(* Logix 5000 project; controller NSH_PLC1 vendor 1 type 14 code 167 rev 32.11; software revision 32.02; part 11 of 12 *)
(* tags used below, declared in another part *)
   Num_Faults : DINT;   // Number of PreCelan Faults
   Num_Warnings : DINT;   // Number of PreCelan Warnings
   Reset_TOF_PRE : DINT;   // Reset pulse duration to Drives
   SpeedIsFactored : BOOL;   // Speed of VFD is factored by Master Speed Factor
   TempAccelerating : BOOL;   // Temp Motor is Accelerating
   TempActive : BOOL;   // Temp Motor is Active
   TempAlarm : BOOL;   // Temp Motor has Alarm
   TempAtSpeed : BOOL;   // Temp Motor is At Speed
   TempCommAlarm : BOOL;   // Temp Motor, AOP communications Alarm
   TempDecelerating : BOOL;   // Temp Motor is Decelerating
   TempFaulted : BOOL;   // Temp Motor is Faulted
   TempMotor : Motor;
   TempReady : BOOL;   // Temp Motor is ready
   TempRunning : BOOL;   // Temp Motor is Running
   TempVFD : VFD_Extra;   // Temp VFD Structure
   BH_FansStarting : BOOL;   // Baghouse 1, 2 or 3 Fans Starting
   CR_LastLine1 : BOOL;   // Last Motor in line 1 Running
   CR_LastLine2 : BOOL;   // Last Motor in line 2 Running
   CR_LastPC1Fan : BOOL;   // Last Motor in Line 1 Fans Running
   CR_LastPC2Fan : BOOL;   // Last Motor in Line 2 Fans Running
   CR_RunCommon : BOOL;   // PreClean, Run Common Units
   CR_RunLine1 : BOOL;   // Pre Clean Run Line 1 Relay
   CR_RunLine2 : BOOL;   // Pre Clean Run Line 2 Relay
   CR_RunPC1_Fans : BOOL;   // Pre Clean Run Line 1 Fans Relay
   CR_RunPC1_FansCO : BOOL;   // Pre Clean Run Line 1 Fans Cleanout Relay
   CR_RunPC2_Fans : BOOL;   // Pre Clean Run Line 2 Fans Relay
   CR_RunPC2_FansCO : BOOL;   // Pre Clean Run Line 2 Fans Cleanout Relay
   CR_StopCommon : BOOL;   // PreClean, Stop Common Units
   CR_StopLine1 : BOOL;   // Pre Clean Stop Line 1 Relay
   CR_StopLine2 : BOOL;   // Pre Clean Stop Line 2 Relay
   DummyVFD : VFD_Extra;   // Dummy
   HS_Starting : BOOL;   // Sheller Sequence is Starting, Prevent Preclean from Starting
   P10_5A : Motor;   // Cross Auger
   P10_5B : Motor;   // Cross Auger
   P10A : Motor;   // Elev to Bins
   P10B : Motor;   // Elev to Bins
   P11A : Motor;   // Line1 Auger
   P11B : Motor;   // Line2 Auger
   P1A : Motor;   // DO Conv.
   P1B : Motor;   // Auger
   P2A : Motor;   // Cross Conv.
   P2B : Motor;   // Stick Reel
   P3A : Motor;   // Stick Reel
   P3B : Motor;   // Stick Reel
   P4A : Motor;   // C. Belt
   P4B : Motor;   // C. Belt
   P5A : Motor;   // Ele. to Vib
   P5B : Motor;   // Ele. to Vib
   P6A : Motor;   // Vib Splitter
   P6B : Motor;   // Vib.Spltr.
   P7A1 : Motor;   // Screener
   P7A2 : Motor;   // Screener
   P7B : Motor;   // Screener
   P7B2_A : Motor;   // Screener
   P7B2_B : Motor;   // Rot.Fdr.
   P8A2_A : Motor;   // Destoner
   P8A2_B : Motor;   // AirLock
   P8A_A : Motor;   // Destoner
   P8A_B : Motor;   // Airlock
   P8B : Motor;   // Destoner
   P8B2_A : Motor;   // Destoner
   P8B2_B : Motor;   // Rot.Fdr.
   P9A : Motor;   // Auger
   P9B : Motor;   // Auger
   PB_StartLine1 : BOOL;   // Pre Clean Start Line 1 Button
   PB_StartLine2 : BOOL;   // Pre Clean Start Line 2 Button
   PB_StopLine1 : BOOL;   // Pre Clean Stop Line 1 Button
   PB_StopLine2 : BOOL;   // Pre Clean Stop Line 2 Button
   PBB1A : Motor;   // AirLock
   PBB1B : Motor;   // Arm
   PBB1C : Motor;   // Cleaning Fan,
   PBB1D : Motor;   // Fan,
   PBB1D_VFD : VFD_Extra;   // Fan
   PBB2A : Motor;   // AirLock
   PBB2B : Motor;   // Arm
   PBB2C : Motor;   // Cleaning Fan,
   PBB2D : Motor;   // Fan,
   PBL_StartLine1 : BOOL;   // Pre Clean Start Line 1 Button Light
   PBL_StartLine2 : BOOL;   // Pre Clean Start Line 2 Button Light
   PBL_StopLine1 : BOOL;   // Pre Clean Stop Line 1 Button Light
   PBL_StopLine2 : BOOL;   // Pre Clean Stop Line 2 Button Light
   PC_AlarmPulseHorn : BOOL;   // PreClean, New Alarm, Pulse Horn
   PC_FaultResetHorn : BOOL;   // PreClean, Fault Reset, sound Horn
   PC_Horn : BOOL;   // PreClean, Horn Output
   PC_LinesStarting : BOOL;   // Pre Clean Line 1 or 2 Starting
   PC_NoEstops : BOOL;   // PreClean, No Estops
   PD1 : Motor;   // Dirt Conv.
   PD2 : Motor;   // Incline
   PR1 : Motor;   // Rock Conv.
   PR2 : Motor;   // Inc. Rock
   PR3 : Motor;   // Belt
   PS1 : Motor;   // Stick Conv.
   PS2 : Motor;   // Inc. Stick Conv.
   PS3 : Motor;   // Twig Conv.
   PS4 : Motor;   // Twig Conv.
   TMR_LineStart1 : TIMER;   // Pre Clean Line 1 Start Warning Timer
   TMR_LineStart2 : TIMER;   // Pre Clean Line 2 Start Warning Timer
   TMR_StartPC1_Fans : TIMER;   // Pre Clean Line 1 Fans Start Warning Timer
   TMR_StartPC1_FansCO : TIMER;   // Pre Clean Line 1 Fans Cleanout Start Warning Timer
   TMR_StartPC2_Fans : TIMER;   // Pre Clean Line 2 Fans Start Warning Timer
   TMR_StartPC2_FansCO : TIMER;   // Pre Clean Line 2 Fans Cleanout Start Warning Timer
(* PreClean, continued *)

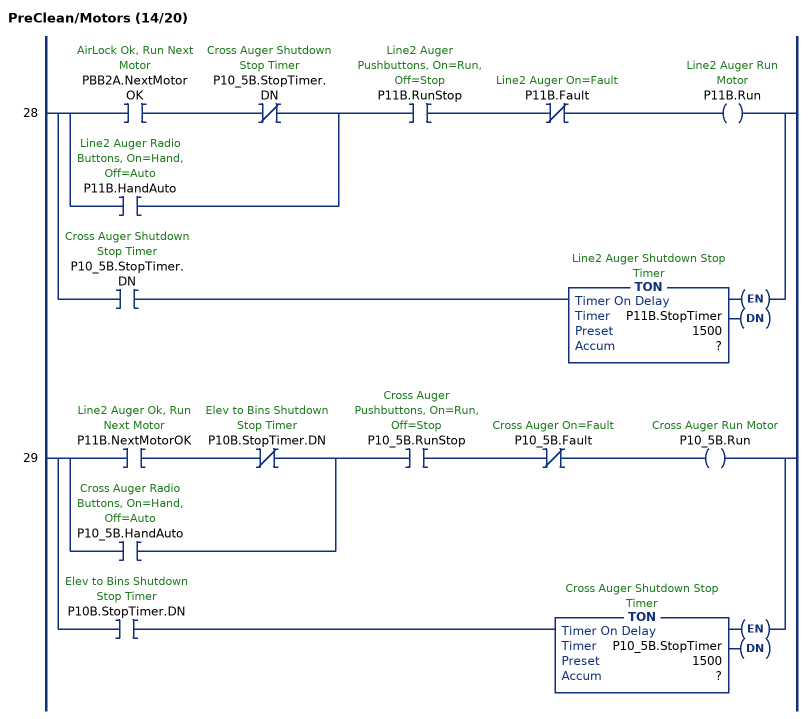
   28: [[XIC(PBB2A.NextMotorOK) XIO(P10_5B.StopTimer.DN) ,XIC(P11B.HandAuto) ] XIC(P11B.RunStop) XIO(P11B.Fault) OTE(P11B.Run) ,XIC(P10_5B.StopTimer.DN) TON(P11B.StopTimer,?,?) ];
   29: [[XIC(P11B.NextMotorOK) XIO(P10B.StopTimer.DN) ,XIC(P10_5B.HandAuto) ] XIC(P10_5B.RunStop) XIO(P10_5B.Fault) OTE(P10_5B.Run) ,XIC(P10B.StopTimer.DN) TON(P10_5B.StopTimer,?,?) ];
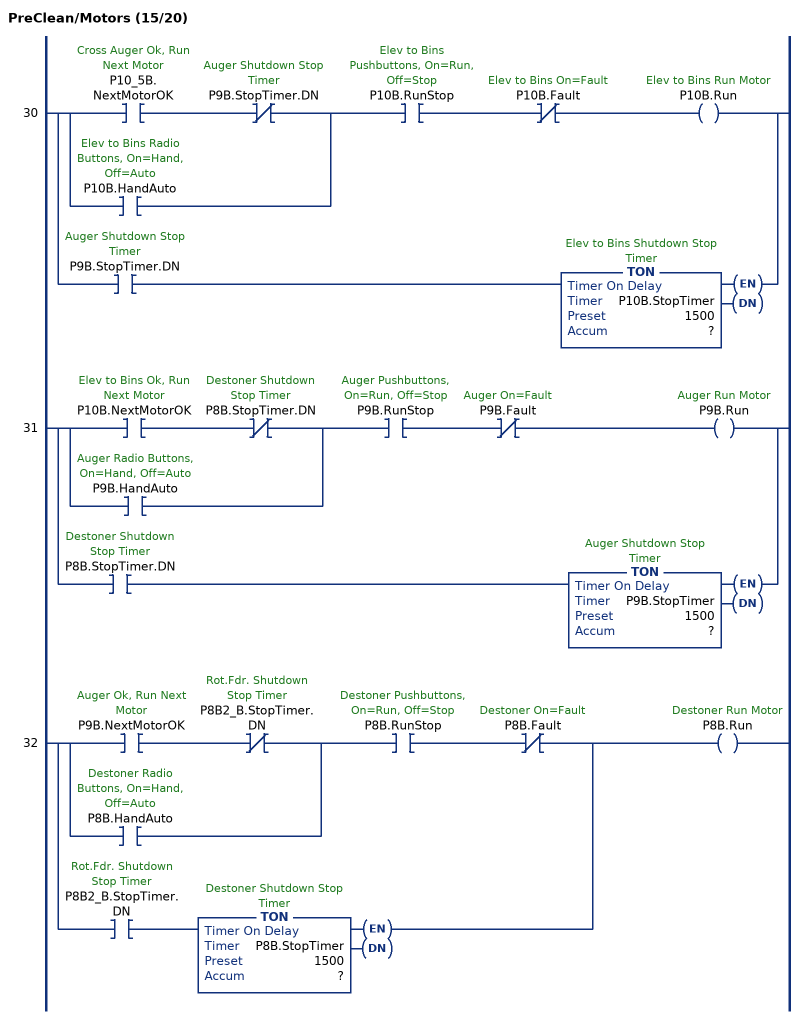
   30: [[XIC(P10_5B.NextMotorOK) XIO(P9B.StopTimer.DN) ,XIC(P10B.HandAuto) ] XIC(P10B.RunStop) XIO(P10B.Fault) OTE(P10B.Run) ,XIC(P9B.StopTimer.DN) TON(P10B.StopTimer,?,?) ];
   31: [[XIC(P10B.NextMotorOK) XIO(P8B.StopTimer.DN) ,XIC(P9B.HandAuto) ] XIC(P9B.RunStop) XIO(P9B.Fault) OTE(P9B.Run) ,XIC(P8B.StopTimer.DN) TON(P9B.StopTimer,?,?) ];
   32: [[XIC(P9B.NextMotorOK) XIO(P8B2_B.StopTimer.DN) ,XIC(P8B.HandAuto) ] XIC(P8B.RunStop) XIO(P8B.Fault) ,XIC(P8B2_B.StopTimer.DN) TON(P8B.StopTimer,?,?) ]OTE(P8B.Run);
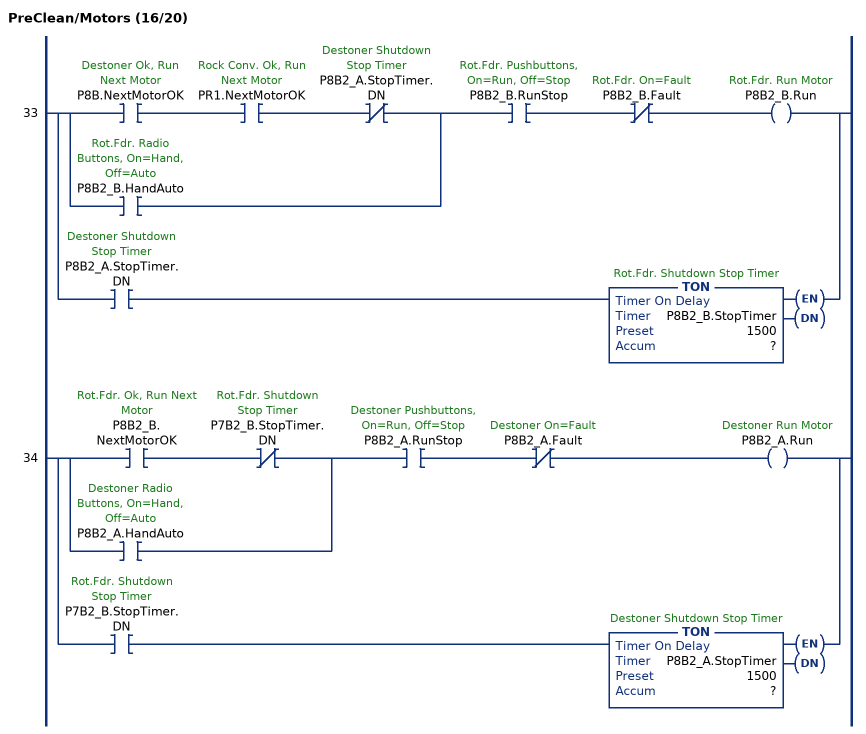
   33: [[XIC(P8B.NextMotorOK) XIC(PR1.NextMotorOK) XIO(P8B2_A.StopTimer.DN) ,XIC(P8B2_B.HandAuto) ] XIC(P8B2_B.RunStop) XIO(P8B2_B.Fault) OTE(P8B2_B.Run) ,XIC(P8B2_A.StopTimer.DN) TON(P8B2_B.StopTimer,?,?) ];
   34: [[XIC(P8B2_B.NextMotorOK) XIO(P7B2_B.StopTimer.DN) ,XIC(P8B2_A.HandAuto) ] XIC(P8B2_A.RunStop) XIO(P8B2_A.Fault) OTE(P8B2_A.Run) ,XIC(P7B2_B.StopTimer.DN) TON(P8B2_A.StopTimer,?,?) ];
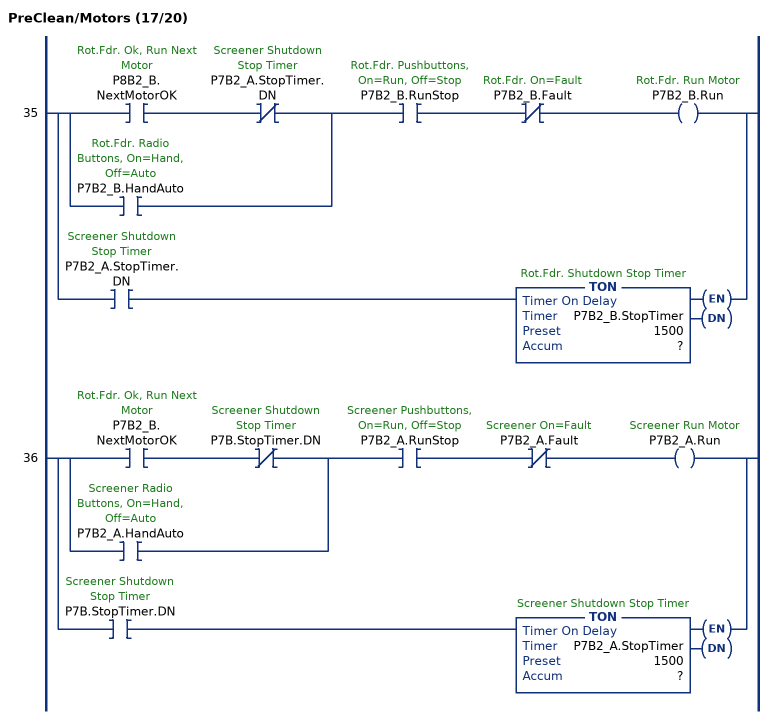
   35: [[XIC(P8B2_B.NextMotorOK) XIO(P7B2_A.StopTimer.DN) ,XIC(P7B2_B.HandAuto) ] XIC(P7B2_B.RunStop) XIO(P7B2_B.Fault) OTE(P7B2_B.Run) ,XIC(P7B2_A.StopTimer.DN) TON(P7B2_B.StopTimer,?,?) ];
   36: [[XIC(P7B2_B.NextMotorOK) XIO(P7B.StopTimer.DN) ,XIC(P7B2_A.HandAuto) ] XIC(P7B2_A.RunStop) XIO(P7B2_A.Fault) OTE(P7B2_A.Run) ,XIC(P7B.StopTimer.DN) TON(P7B2_A.StopTimer,?,?) ];
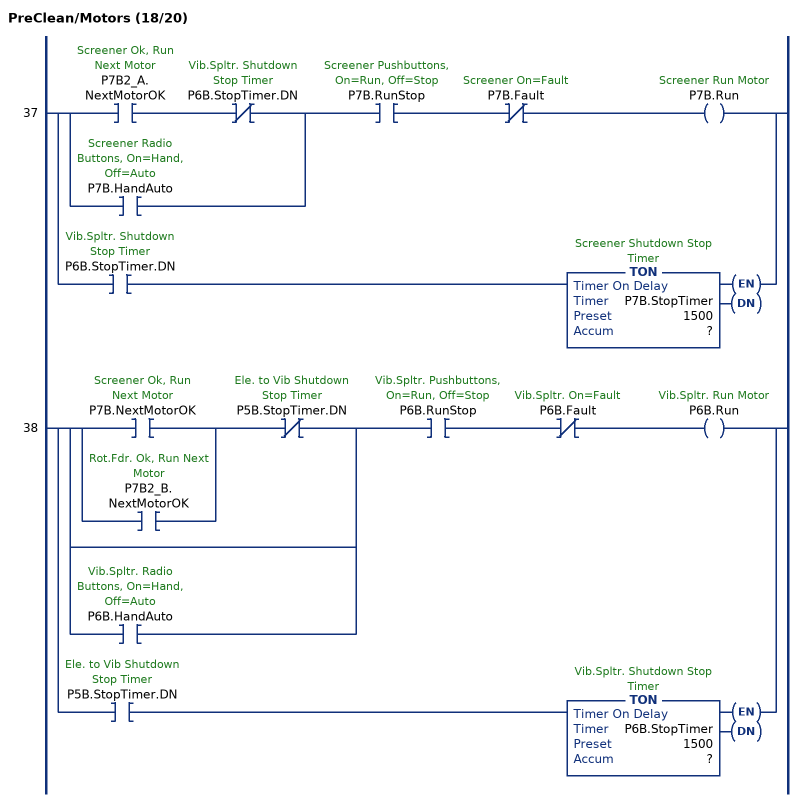
   37: [[XIC(P7B2_A.NextMotorOK) XIO(P6B.StopTimer.DN) ,XIC(P7B.HandAuto) ] XIC(P7B.RunStop) XIO(P7B.Fault) OTE(P7B.Run) ,XIC(P6B.StopTimer.DN) TON(P7B.StopTimer,?,?) ];
   38: [[[XIC(P7B.NextMotorOK) ,XIC(P7B2_B.NextMotorOK) ] XIO(P5B.StopTimer.DN) ,,XIC(P6B.HandAuto) ] XIC(P6B.RunStop) XIO(P6B.Fault) OTE(P6B.Run) ,XIC(P5B.StopTimer.DN) TON(P6B.StopTimer,?,?) ];
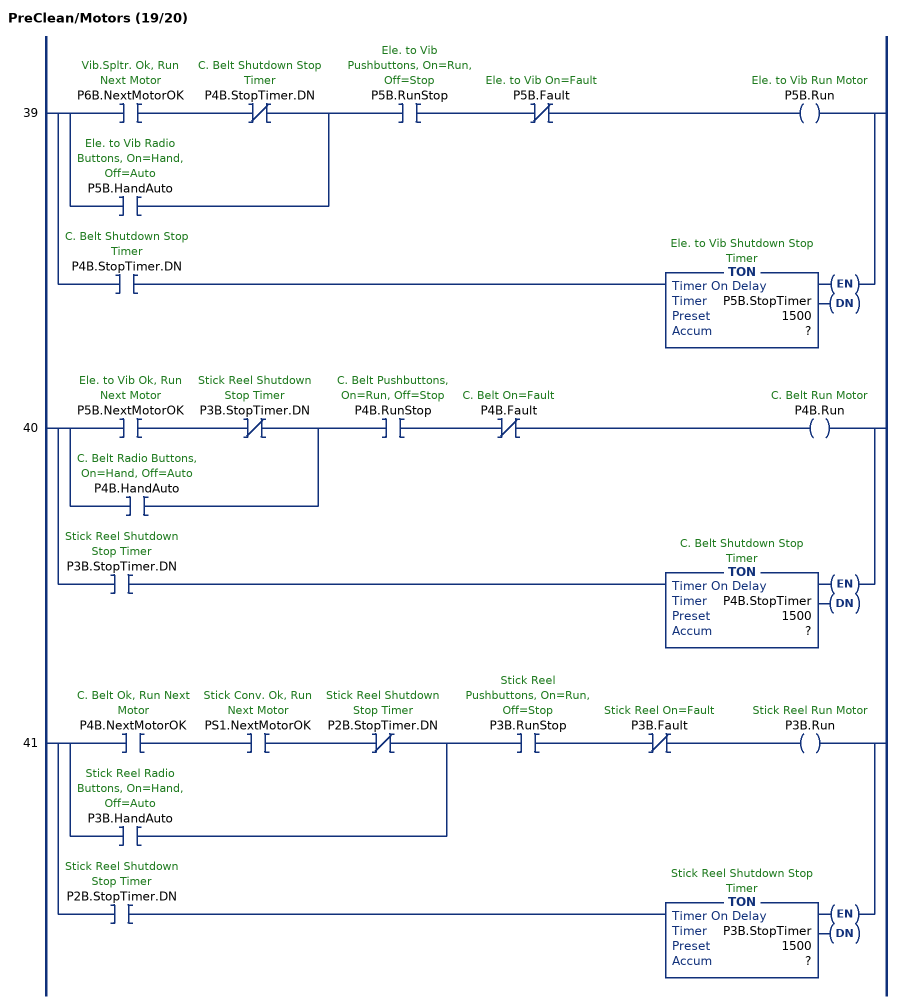
   39: [[XIC(P6B.NextMotorOK) XIO(P4B.StopTimer.DN) ,XIC(P5B.HandAuto) ] XIC(P5B.RunStop) XIO(P5B.Fault) OTE(P5B.Run) ,XIC(P4B.StopTimer.DN) TON(P5B.StopTimer,?,?) ];
   40: [[XIC(P5B.NextMotorOK) XIO(P3B.StopTimer.DN) ,XIC(P4B.HandAuto) ] XIC(P4B.RunStop) XIO(P4B.Fault) OTE(P4B.Run) ,XIC(P3B.StopTimer.DN) TON(P4B.StopTimer,?,?) ];
   41: [[XIC(P4B.NextMotorOK) XIC(PS1.NextMotorOK) XIO(P2B.StopTimer.DN) ,XIC(P3B.HandAuto) ] XIC(P3B.RunStop) XIO(P3B.Fault) OTE(P3B.Run) ,XIC(P2B.StopTimer.DN) TON(P3B.StopTimer,?,?) ];
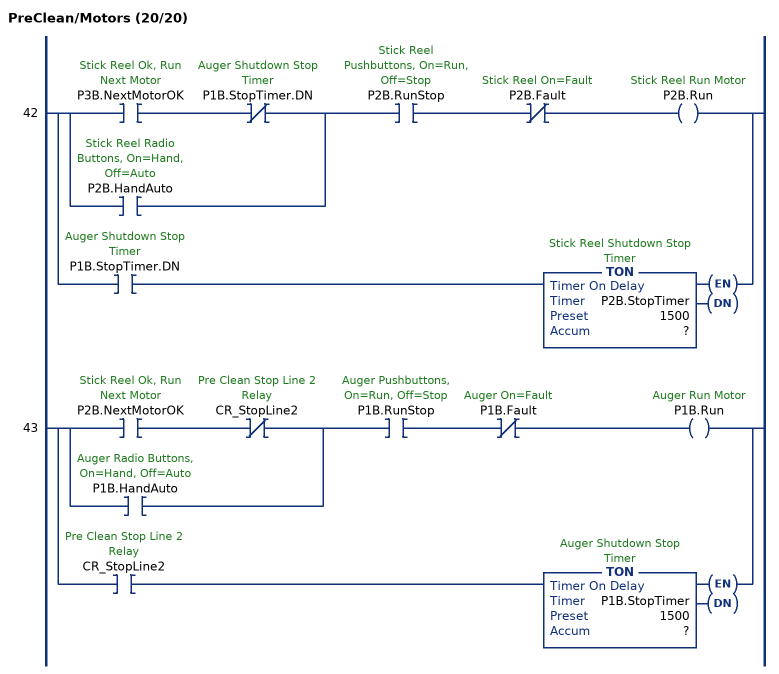
   42: [[XIC(P3B.NextMotorOK) XIO(P1B.StopTimer.DN) ,XIC(P2B.HandAuto) ] XIC(P2B.RunStop) XIO(P2B.Fault) OTE(P2B.Run) ,XIC(P1B.StopTimer.DN) TON(P2B.StopTimer,?,?) ];
   43: [[XIC(P2B.NextMotorOK) XIO(CR_StopLine2) ,XIC(P1B.HandAuto) ] XIC(P1B.RunStop) XIO(P1B.Fault) OTE(P1B.Run) ,XIC(CR_StopLine2) TON(P1B.StopTimer,?,?) ];
END_ROUTINE

ROUTINE MotorStatusSUB   (* ladder *)
// Update Status Subroutine
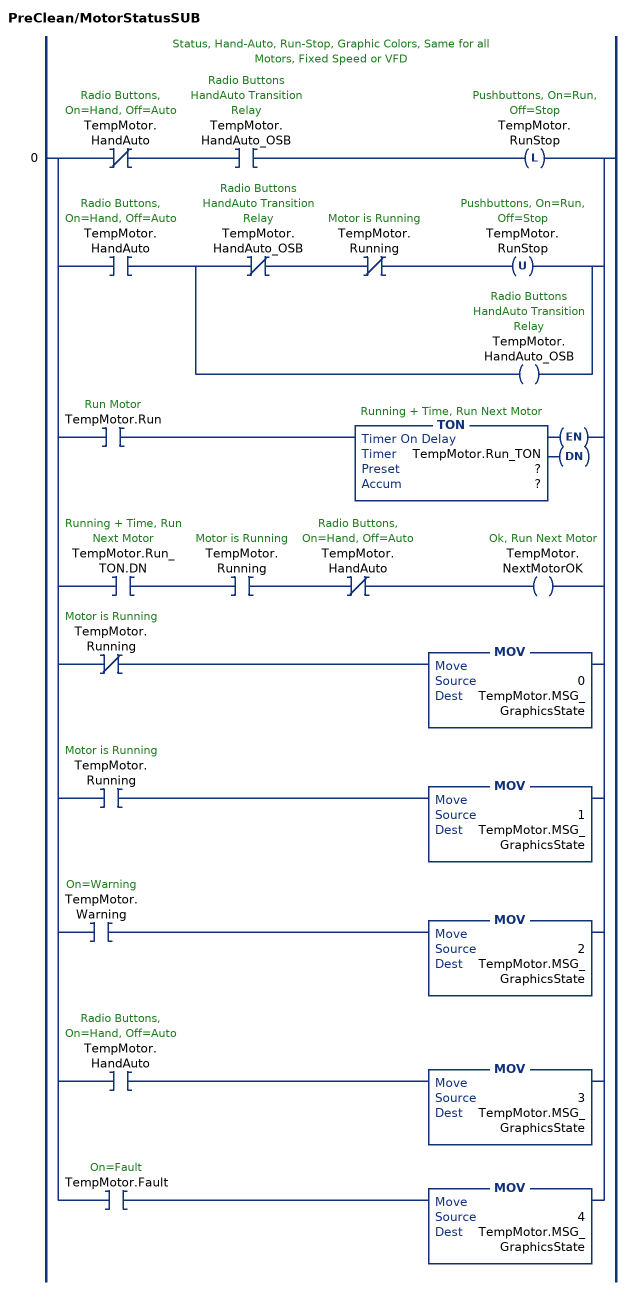
   // Status, Hand-Auto, Run-Stop, Graphic Colors, Same for all
   // Motors, Fixed Speed or VFD
   0: [XIO(TempMotor.HandAuto) XIC(TempMotor.HandAuto_OSB) OTL(TempMotor.RunStop) ,XIC(TempMotor.HandAuto) [XIO(TempMotor.HandAuto_OSB) XIO(TempMotor.Running) OTU(TempMotor.RunStop) ,OTE(TempMotor.HandAuto_OSB) ] ,XIC(TempMotor.Run) TON(TempMotor.Run_TON,?,?) ,XIC(TempMotor.Run_TON.DN) XIC(TempMotor.Running) XIO(TempMotor.HandAuto) OTE(TempMotor.NextMotorOK) ,XIO(TempMotor.Running) MOV(0,TempMotor.MSG_GraphicsState) ,XIC(TempMotor.Running) MOV(1,TempMotor.MSG_GraphicsState) ,XIC(TempMotor.Warning) MOV(2,TempMotor.MSG_GraphicsState) ,XIC(TempMotor.HandAuto) MOV(3,TempMotor.MSG_GraphicsState) ,XIC(TempMotor.Fault) MOV(4,TempMotor.MSG_GraphicsState) ];
END_ROUTINE

ROUTINE PC_MainJSR   (* ladder *)
// Jump To Other Routines
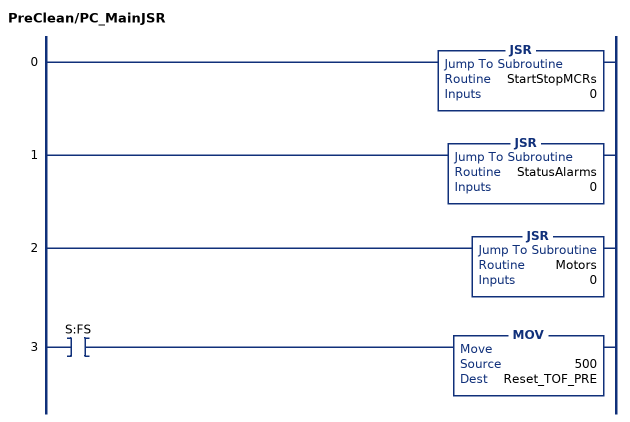
   0: JSR(StartStopMCRs,0);
   1: JSR(StatusAlarms,0);
   2: JSR(Motors,0);
   3: XIC(S:FS)MOV(500,Reset_TOF_PRE);
END_ROUTINE

ROUTINE PF525_StatusAlmWarnSUB   (* ladder *)
// Decode Status Bits and Set Warnings and Alarm for PowerFlex525
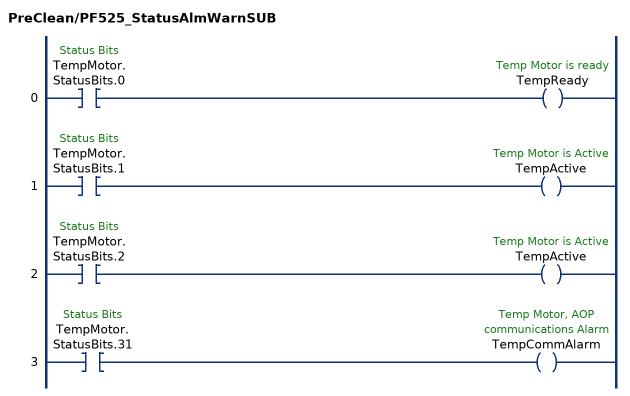
   0: XIC(TempMotor.StatusBits.0)OTE(TempReady);
   1: XIC(TempMotor.StatusBits.1)OTE(TempActive);
   2: XIC(TempMotor.StatusBits.2)OTE(TempActive);
   3: XIC(TempMotor.StatusBits.31)OTE(TempCommAlarm);
END_ROUTINE

ROUTINE PF755_StatusAlmWarnSUB   (* ladder *)
// Decode Status Bits and Set Warnings and Alarm for PowerFlex755
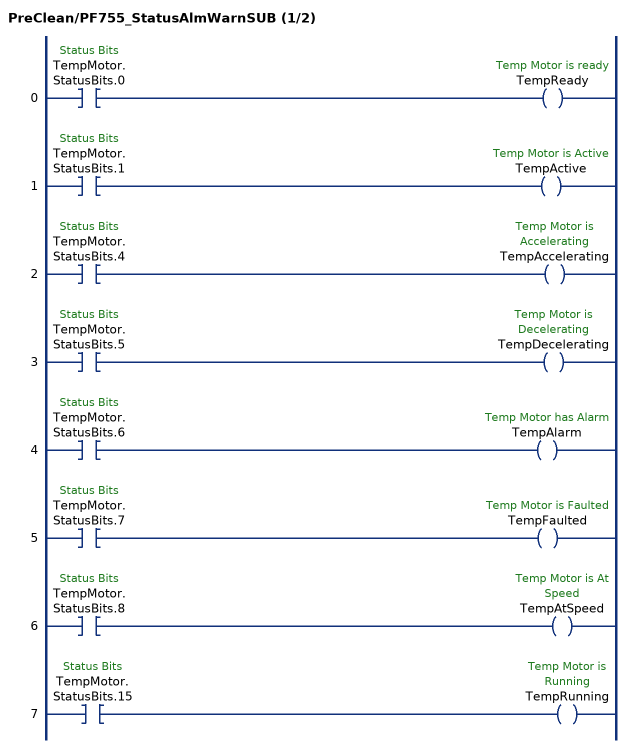
   0: XIC(TempMotor.StatusBits.0)OTE(TempReady);
   1: XIC(TempMotor.StatusBits.1)OTE(TempActive);
   2: XIC(TempMotor.StatusBits.4)OTE(TempAccelerating);
   3: XIC(TempMotor.StatusBits.5)OTE(TempDecelerating);
   4: XIC(TempMotor.StatusBits.6)OTE(TempAlarm);
   5: XIC(TempMotor.StatusBits.7)OTE(TempFaulted);
   6: XIC(TempMotor.StatusBits.8)OTE(TempAtSpeed);
   7: XIC(TempMotor.StatusBits.15)OTE(TempRunning);
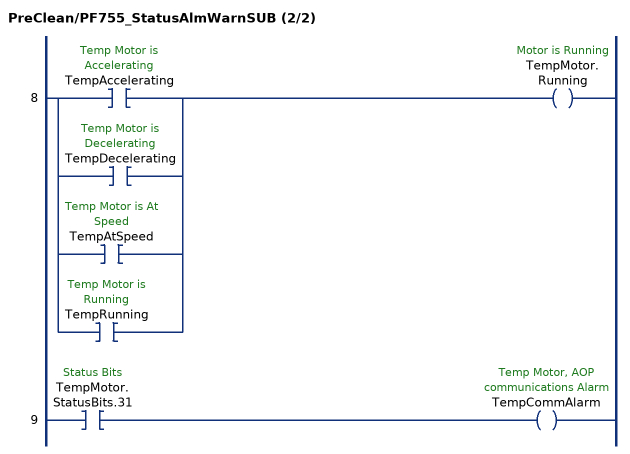
   8: [XIC(TempAccelerating) ,XIC(TempDecelerating) ,XIC(TempAtSpeed) ,XIC(TempRunning) ]OTE(TempMotor.Running);
   9: XIC(TempMotor.StatusBits.31)OTE(TempCommAlarm);
END_ROUTINE

ROUTINE StartStopMCRs   (* ladder *)
// Precleaner Logic
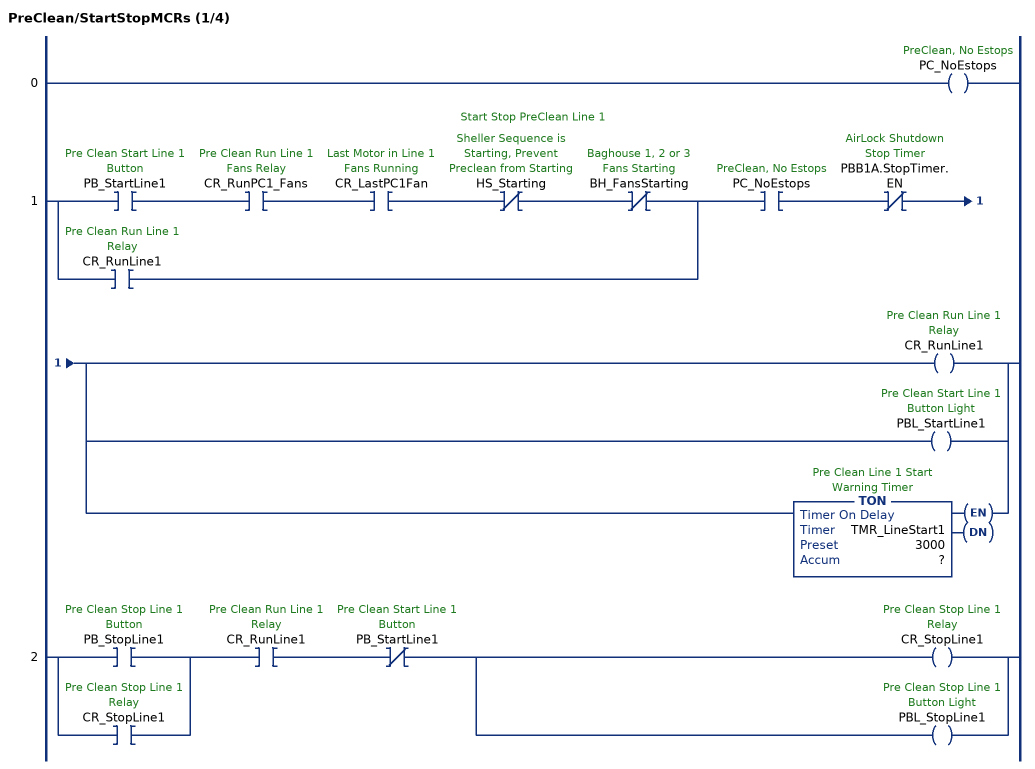
   0: OTE(PC_NoEstops);
   // Start Stop PreClean Line 1
   1: [XIC(PB_StartLine1) XIC(CR_RunPC1_Fans) XIC(CR_LastPC1Fan) XIO(HS_Starting) XIO(BH_FansStarting) ,XIC(CR_RunLine1) ]XIC(PC_NoEstops)XIO(PBB1A.StopTimer.EN)[OTE(CR_RunLine1) ,OTE(PBL_StartLine1) ,TON(TMR_LineStart1,?,?) ];
   2: [XIC(PB_StopLine1) ,XIC(CR_StopLine1) ]XIC(CR_RunLine1)XIO(PB_StartLine1)[OTE(CR_StopLine1) ,OTE(PBL_StopLine1) ];
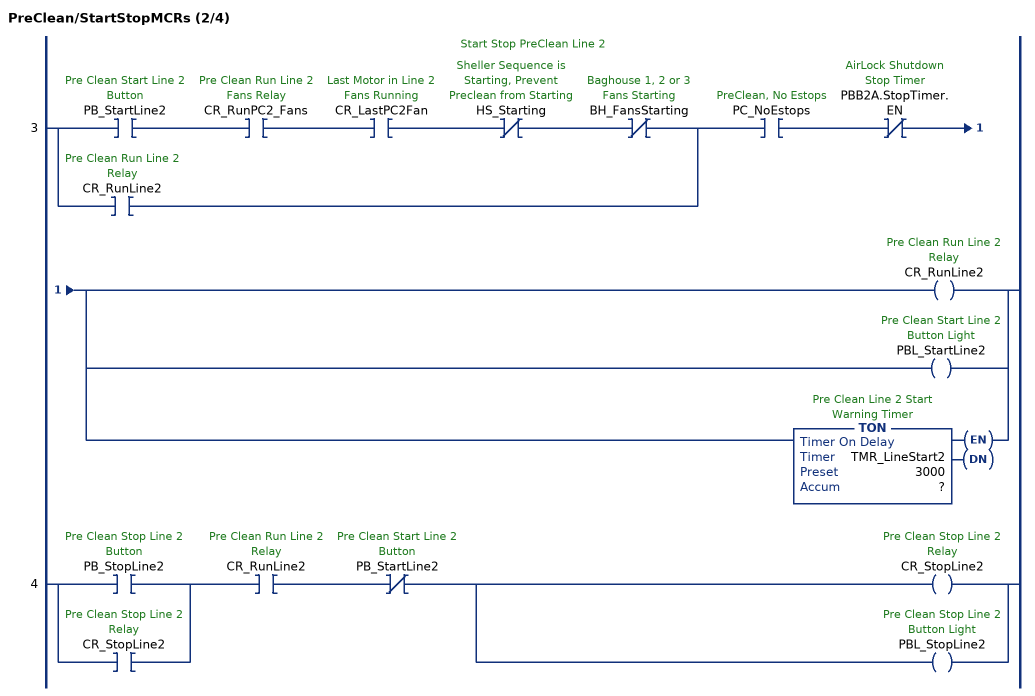
   // Start Stop PreClean Line 2
   3: [XIC(PB_StartLine2) XIC(CR_RunPC2_Fans) XIC(CR_LastPC2Fan) XIO(HS_Starting) XIO(BH_FansStarting) ,XIC(CR_RunLine2) ]XIC(PC_NoEstops)XIO(PBB2A.StopTimer.EN)[OTE(CR_RunLine2) ,OTE(PBL_StartLine2) ,TON(TMR_LineStart2,?,?) ];
   4: [XIC(PB_StopLine2) ,XIC(CR_StopLine2) ]XIC(CR_RunLine2)XIO(PB_StartLine2)[OTE(CR_StopLine2) ,OTE(PBL_StopLine2) ];
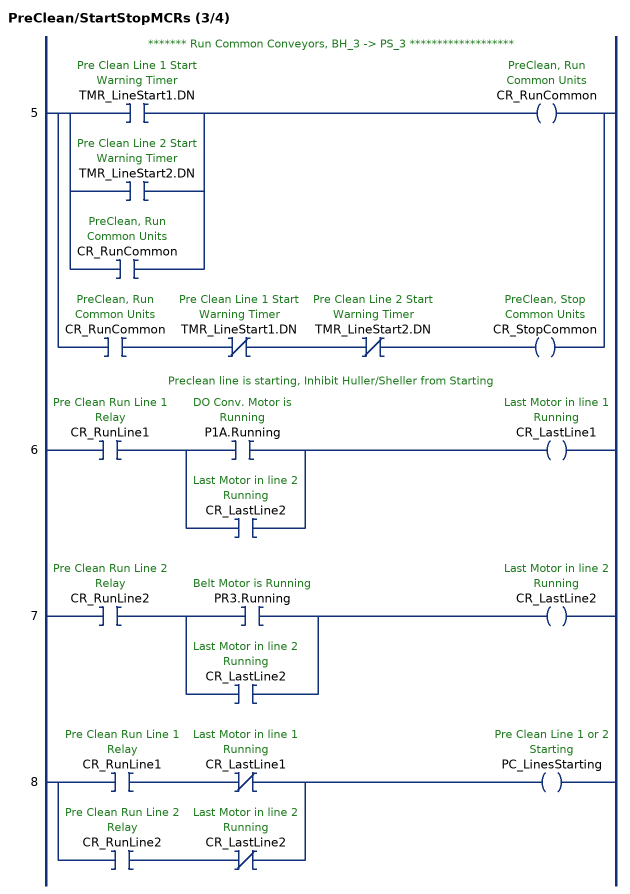
   // ******* Run Common Conveyors, BH_3 -> PS_3 *******************
   5: [[XIC(TMR_LineStart1.DN) ,XIC(TMR_LineStart2.DN) ,XIC(CR_RunCommon) ] OTE(CR_RunCommon) ,XIC(CR_RunCommon) XIO(TMR_LineStart1.DN) XIO(TMR_LineStart2.DN) OTE(CR_StopCommon) ];
   // Preclean line is starting, Inhibit Huller/Sheller from Starting
   6: XIC(CR_RunLine1)[XIC(P1A.Running) ,XIC(CR_LastLine2) ]OTE(CR_LastLine1);
   7: XIC(CR_RunLine2)[XIC(PR3.Running) ,XIC(CR_LastLine2) ]OTE(CR_LastLine2);
   8: [XIC(CR_RunLine1) XIO(CR_LastLine1) ,XIC(CR_RunLine2) XIO(CR_LastLine2) ]OTE(PC_LinesStarting);
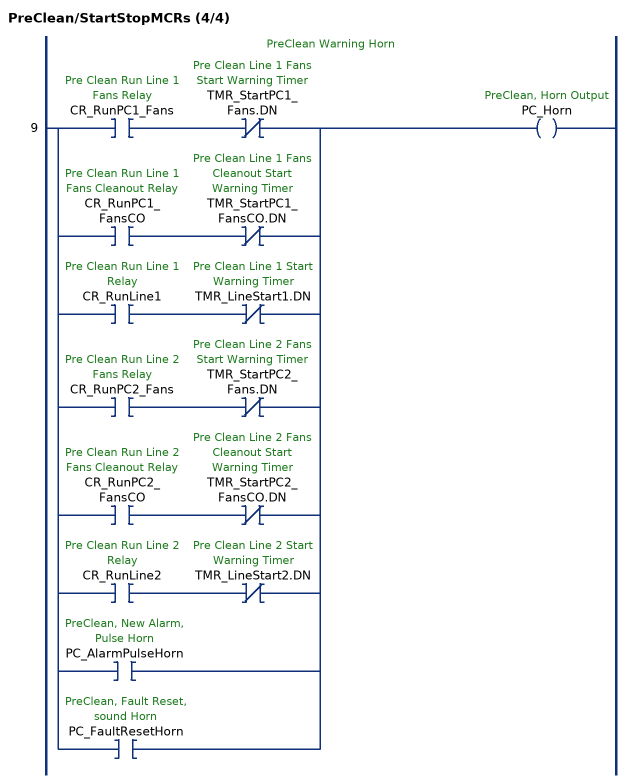
   // PreClean Warning Horn
   9: [XIC(CR_RunPC1_Fans) XIO(TMR_StartPC1_Fans.DN) ,XIC(CR_RunPC1_FansCO) XIO(TMR_StartPC1_FansCO.DN) ,XIC(CR_RunLine1) XIO(TMR_LineStart1.DN) ,XIC(CR_RunPC2_Fans) XIO(TMR_StartPC2_Fans.DN) ,XIC(CR_RunPC2_FansCO) XIO(TMR_StartPC2_FansCO.DN) ,XIC(CR_RunLine2) XIO(TMR_LineStart2.DN) ,XIC(PC_AlarmPulseHorn) ,XIC(PC_FaultResetHorn) ]OTE(PC_Horn);
END_ROUTINE

ROUTINE StatusAlarms   (* ladder *)
// Motor Status And Alarms
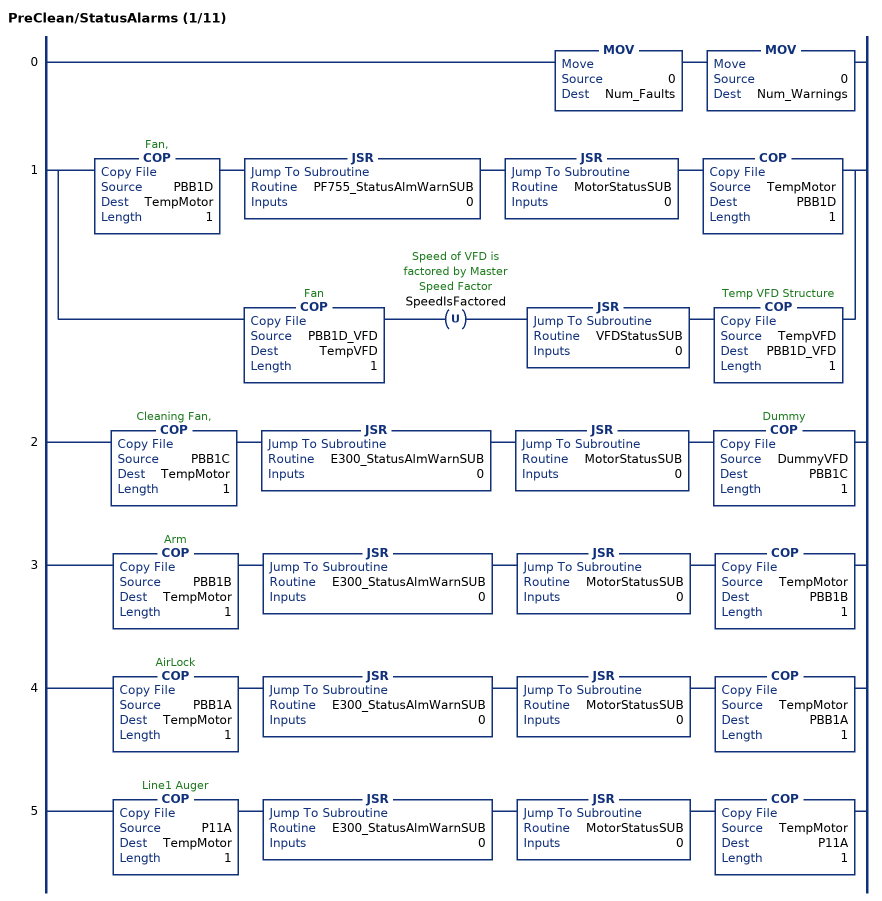
   0: MOV(0,Num_Faults)MOV(0,Num_Warnings);
   1: [COP(PBB1D,TempMotor,1) JSR(PF755_StatusAlmWarnSUB,0) JSR(MotorStatusSUB,0) COP(TempMotor,PBB1D,1) ,COP(PBB1D_VFD,TempVFD,1) OTU(SpeedIsFactored) JSR(VFDStatusSUB,0) COP(TempVFD,PBB1D_VFD,1) ];
   2: COP(PBB1C,TempMotor,1)JSR(E300_StatusAlmWarnSUB,0)JSR(MotorStatusSUB,0)COP(DummyVFD,PBB1C,1);
   3: COP(PBB1B,TempMotor,1)JSR(E300_StatusAlmWarnSUB,0)JSR(MotorStatusSUB,0)COP(TempMotor,PBB1B,1);
   4: COP(PBB1A,TempMotor,1)JSR(E300_StatusAlmWarnSUB,0)JSR(MotorStatusSUB,0)COP(TempMotor,PBB1A,1);
   5: COP(P11A,TempMotor,1)JSR(E300_StatusAlmWarnSUB,0)JSR(MotorStatusSUB,0)COP(TempMotor,P11A,1);
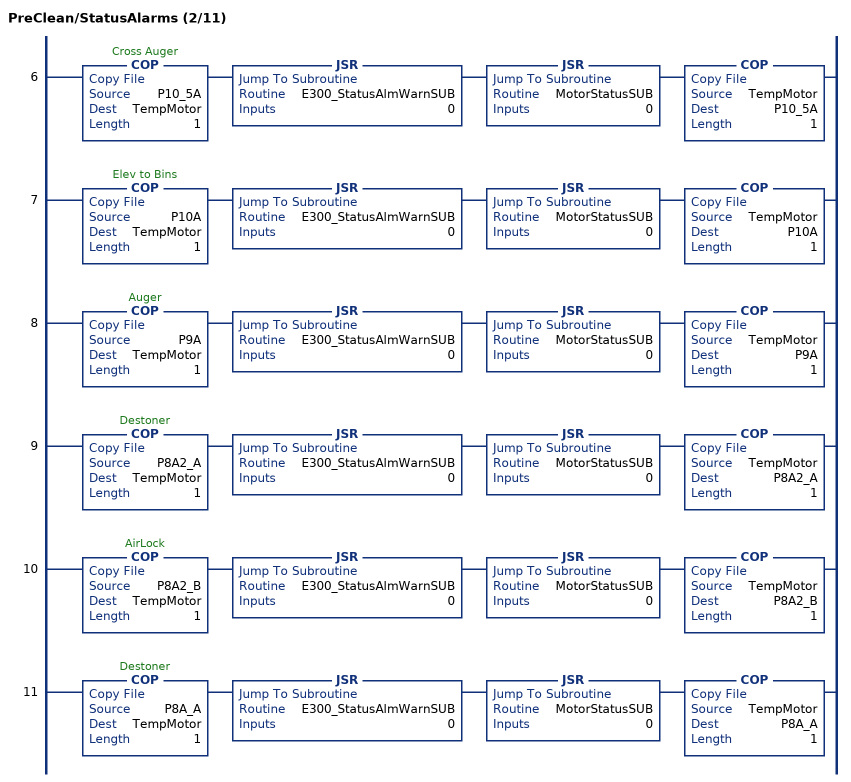
   6: COP(P10_5A,TempMotor,1)JSR(E300_StatusAlmWarnSUB,0)JSR(MotorStatusSUB,0)COP(TempMotor,P10_5A,1);
   7: COP(P10A,TempMotor,1)JSR(E300_StatusAlmWarnSUB,0)JSR(MotorStatusSUB,0)COP(TempMotor,P10A,1);
   8: COP(P9A,TempMotor,1)JSR(E300_StatusAlmWarnSUB,0)JSR(MotorStatusSUB,0)COP(TempMotor,P9A,1);
   9: COP(P8A2_A,TempMotor,1)JSR(E300_StatusAlmWarnSUB,0)JSR(MotorStatusSUB,0)COP(TempMotor,P8A2_A,1);
   10: COP(P8A2_B,TempMotor,1)JSR(E300_StatusAlmWarnSUB,0)JSR(MotorStatusSUB,0)COP(TempMotor,P8A2_B,1);
   11: COP(P8A_A,TempMotor,1)JSR(E300_StatusAlmWarnSUB,0)JSR(MotorStatusSUB,0)COP(TempMotor,P8A_A,1);
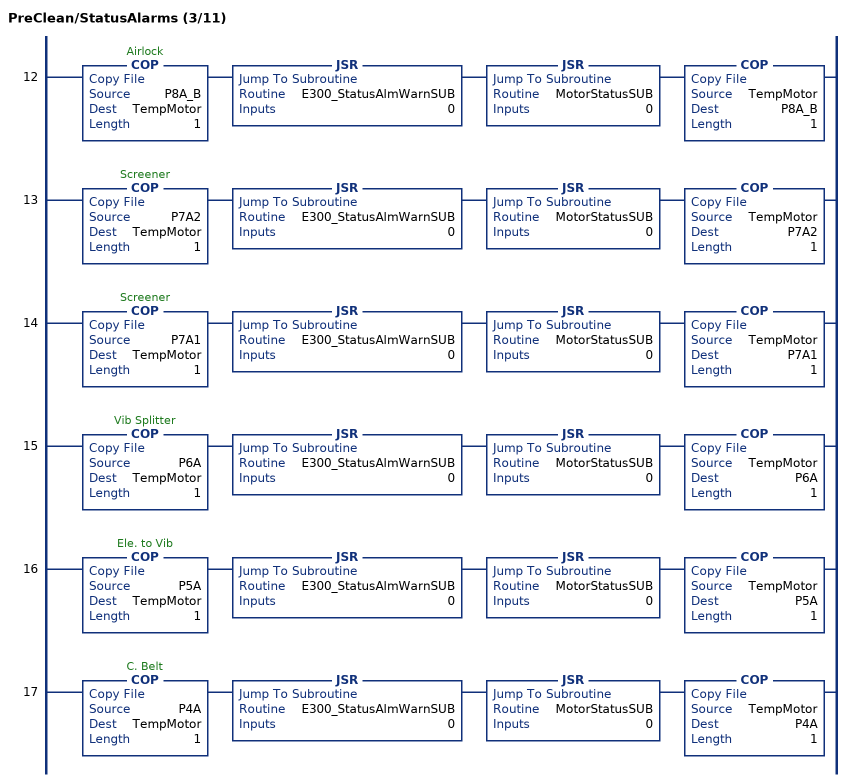
   12: COP(P8A_B,TempMotor,1)JSR(E300_StatusAlmWarnSUB,0)JSR(MotorStatusSUB,0)COP(TempMotor,P8A_B,1);
   13: COP(P7A2,TempMotor,1)JSR(E300_StatusAlmWarnSUB,0)JSR(MotorStatusSUB,0)COP(TempMotor,P7A2,1);
   14: COP(P7A1,TempMotor,1)JSR(E300_StatusAlmWarnSUB,0)JSR(MotorStatusSUB,0)COP(TempMotor,P7A1,1);
   15: COP(P6A,TempMotor,1)JSR(E300_StatusAlmWarnSUB,0)JSR(MotorStatusSUB,0)COP(TempMotor,P6A,1);
   16: COP(P5A,TempMotor,1)JSR(E300_StatusAlmWarnSUB,0)JSR(MotorStatusSUB,0)COP(TempMotor,P5A,1);
   17: COP(P4A,TempMotor,1)JSR(E300_StatusAlmWarnSUB,0)JSR(MotorStatusSUB,0)COP(TempMotor,P4A,1);
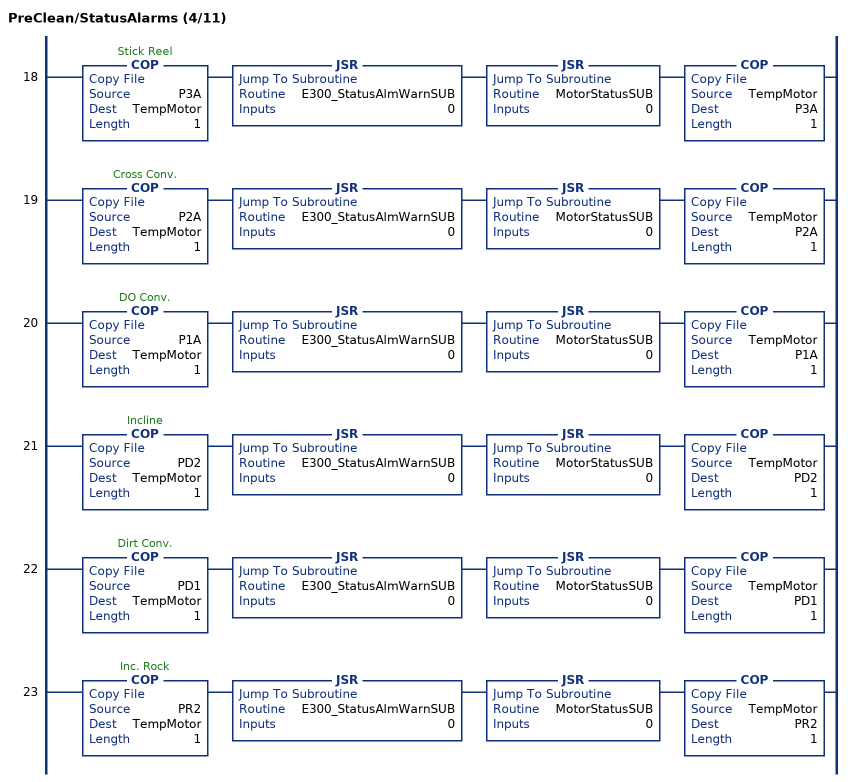
   18: COP(P3A,TempMotor,1)JSR(E300_StatusAlmWarnSUB,0)JSR(MotorStatusSUB,0)COP(TempMotor,P3A,1);
   19: COP(P2A,TempMotor,1)JSR(E300_StatusAlmWarnSUB,0)JSR(MotorStatusSUB,0)COP(TempMotor,P2A,1);
   20: COP(P1A,TempMotor,1)JSR(E300_StatusAlmWarnSUB,0)JSR(MotorStatusSUB,0)COP(TempMotor,P1A,1);
   21: COP(PD2,TempMotor,1)JSR(E300_StatusAlmWarnSUB,0)JSR(MotorStatusSUB,0)COP(TempMotor,PD2,1);
   22: COP(PD1,TempMotor,1)JSR(E300_StatusAlmWarnSUB,0)JSR(MotorStatusSUB,0)COP(TempMotor,PD1,1);
   23: COP(PR2,TempMotor,1)JSR(E300_StatusAlmWarnSUB,0)JSR(MotorStatusSUB,0)COP(TempMotor,PR2,1);
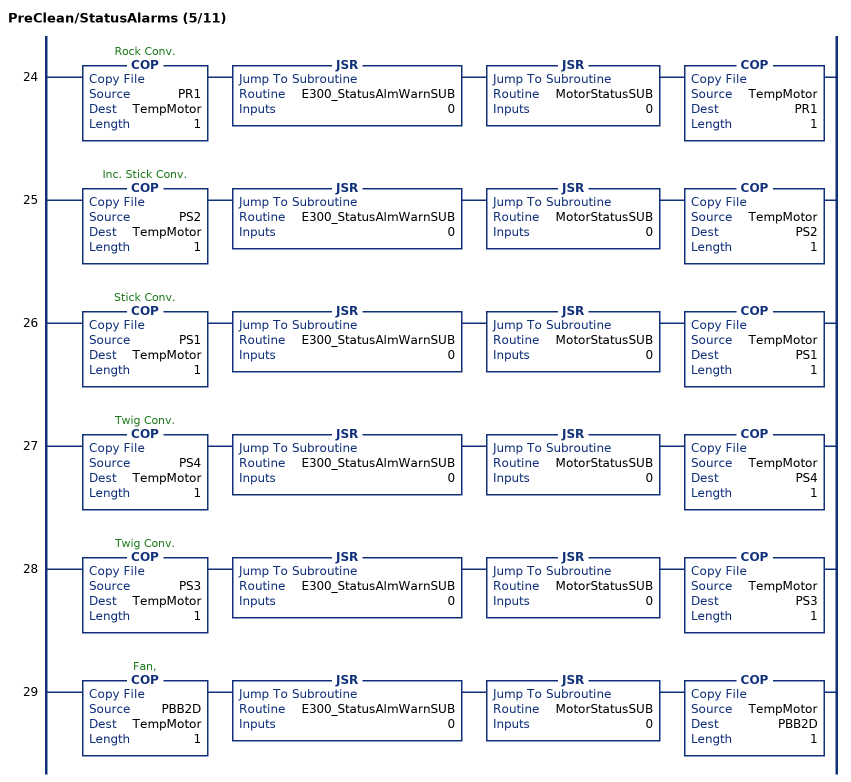
   24: COP(PR1,TempMotor,1)JSR(E300_StatusAlmWarnSUB,0)JSR(MotorStatusSUB,0)COP(TempMotor,PR1,1);
   25: COP(PS2,TempMotor,1)JSR(E300_StatusAlmWarnSUB,0)JSR(MotorStatusSUB,0)COP(TempMotor,PS2,1);
   26: COP(PS1,TempMotor,1)JSR(E300_StatusAlmWarnSUB,0)JSR(MotorStatusSUB,0)COP(TempMotor,PS1,1);
   27: COP(PS4,TempMotor,1)JSR(E300_StatusAlmWarnSUB,0)JSR(MotorStatusSUB,0)COP(TempMotor,PS4,1);
   28: COP(PS3,TempMotor,1)JSR(E300_StatusAlmWarnSUB,0)JSR(MotorStatusSUB,0)COP(TempMotor,PS3,1);
   29: COP(PBB2D,TempMotor,1)JSR(E300_StatusAlmWarnSUB,0)JSR(MotorStatusSUB,0)COP(TempMotor,PBB2D,1);
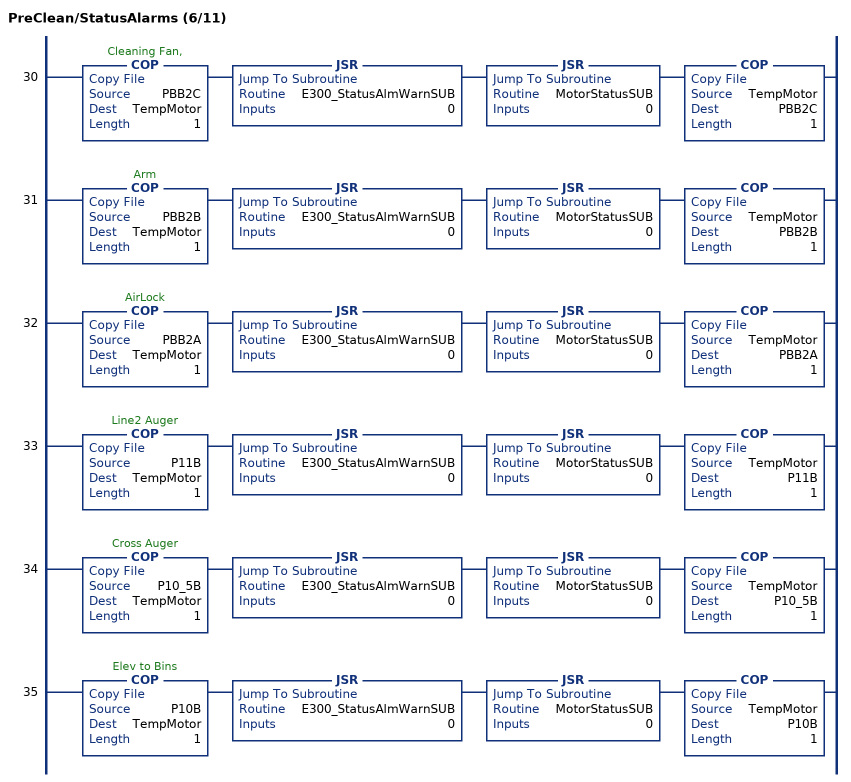
   30: COP(PBB2C,TempMotor,1)JSR(E300_StatusAlmWarnSUB,0)JSR(MotorStatusSUB,0)COP(TempMotor,PBB2C,1);
   31: COP(PBB2B,TempMotor,1)JSR(E300_StatusAlmWarnSUB,0)JSR(MotorStatusSUB,0)COP(TempMotor,PBB2B,1);
   32: COP(PBB2A,TempMotor,1)JSR(E300_StatusAlmWarnSUB,0)JSR(MotorStatusSUB,0)COP(TempMotor,PBB2A,1);
   33: COP(P11B,TempMotor,1)JSR(E300_StatusAlmWarnSUB,0)JSR(MotorStatusSUB,0)COP(TempMotor,P11B,1);
   34: COP(P10_5B,TempMotor,1)JSR(E300_StatusAlmWarnSUB,0)JSR(MotorStatusSUB,0)COP(TempMotor,P10_5B,1);
   35: COP(P10B,TempMotor,1)JSR(E300_StatusAlmWarnSUB,0)JSR(MotorStatusSUB,0)COP(TempMotor,P10B,1);
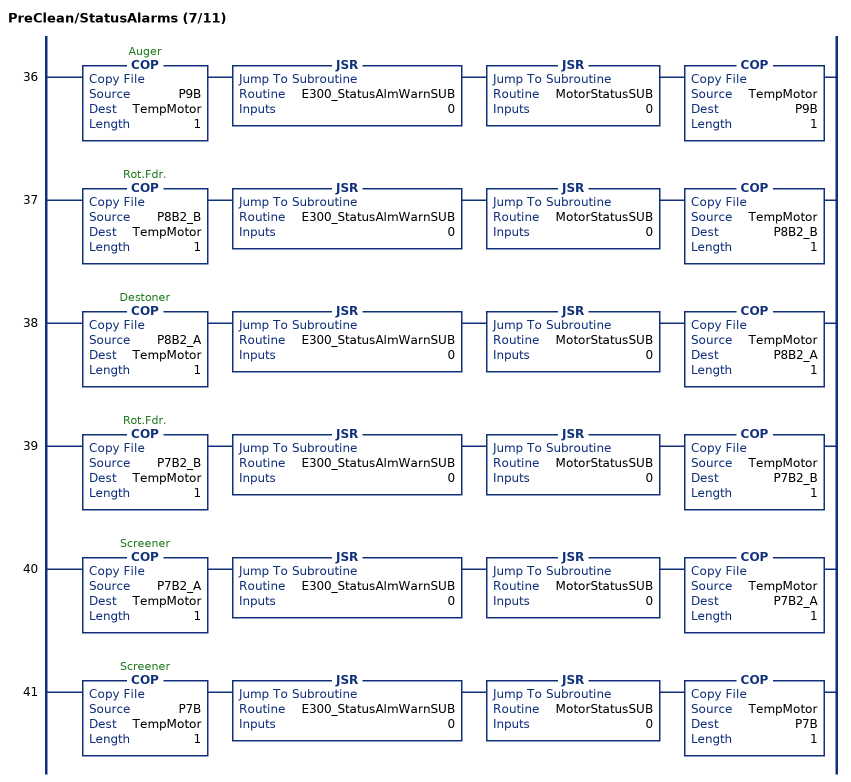
   36: COP(P9B,TempMotor,1)JSR(E300_StatusAlmWarnSUB,0)JSR(MotorStatusSUB,0)COP(TempMotor,P9B,1);
   37: COP(P8B2_B,TempMotor,1)JSR(E300_StatusAlmWarnSUB,0)JSR(MotorStatusSUB,0)COP(TempMotor,P8B2_B,1);
   38: COP(P8B2_A,TempMotor,1)JSR(E300_StatusAlmWarnSUB,0)JSR(MotorStatusSUB,0)COP(TempMotor,P8B2_A,1);
   39: COP(P7B2_B,TempMotor,1)JSR(E300_StatusAlmWarnSUB,0)JSR(MotorStatusSUB,0)COP(TempMotor,P7B2_B,1);
   40: COP(P7B2_A,TempMotor,1)JSR(E300_StatusAlmWarnSUB,0)JSR(MotorStatusSUB,0)COP(TempMotor,P7B2_A,1);
   41: COP(P7B,TempMotor,1)JSR(E300_StatusAlmWarnSUB,0)JSR(MotorStatusSUB,0)COP(TempMotor,P7B,1);
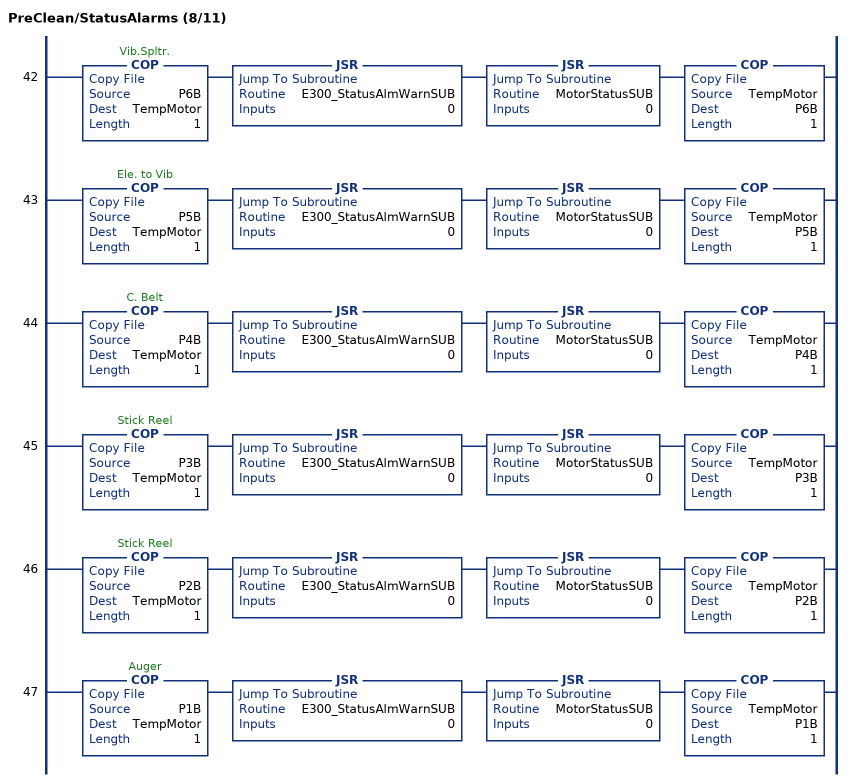
   42: COP(P6B,TempMotor,1)JSR(E300_StatusAlmWarnSUB,0)JSR(MotorStatusSUB,0)COP(TempMotor,P6B,1);
   43: COP(P5B,TempMotor,1)JSR(E300_StatusAlmWarnSUB,0)JSR(MotorStatusSUB,0)COP(TempMotor,P5B,1);
   44: COP(P4B,TempMotor,1)JSR(E300_StatusAlmWarnSUB,0)JSR(MotorStatusSUB,0)COP(TempMotor,P4B,1);
   45: COP(P3B,TempMotor,1)JSR(E300_StatusAlmWarnSUB,0)JSR(MotorStatusSUB,0)COP(TempMotor,P3B,1);
   46: COP(P2B,TempMotor,1)JSR(E300_StatusAlmWarnSUB,0)JSR(MotorStatusSUB,0)COP(TempMotor,P2B,1);
   47: COP(P1B,TempMotor,1)JSR(E300_StatusAlmWarnSUB,0)JSR(MotorStatusSUB,0)COP(TempMotor,P1B,1);
